(* PLC project Generated.project, CODESYS CODESYS V3.5 SP19 Patch 1 *)
(* stored: creationDateTime 2026-08-18T15:58:33.203512, modificationDateTime 2026-08-18T15:58:33.203512 *)

(* ======================================================================= 🔄 ST_ChainCycleSemiAuto — Diagnostic chronologique Séquenceur Semi-Auto ─────────────────────────────────────────────────────────────── 🎯 Rôle : Vue dépannage / Watch CODESYS pour le cycle semi-automatique 📄 Doc métier : DOC/AF/AF_Partie-14_Fonction_Troubleshooting/FB_TroubleshootingView_v1.2.md 🔒 Sécurité : 100% lecture seule / diagnostic d'observation ======================================================================= *)
TYPE ST_ChainCycleSemiAuto : STRUCT
  Idx101_ModeSemiAutoActive : BOOL;  (* 🚦 1. Conditions d'engagement et autorisations 1 = Mode arbitré SEMI_AUTO actif | 0 = Autre mode *)
  Idx102_PowerAndSafetyOk : BOOL;  (* 1 = Chaîne de sécurité OK (PowerContactorEngaged) *)
  Idx103_HeartbeatIhmOk : BOOL;  (* 1 = Liaison IHM<->PLC valide *)
  Idx104_DeadmanArmed : BOOL;  (* 1 = Bouton homme-mort armé (fenêtre 3s active) *)
  Idx105_MancheDeflechi : BOOL;  (* 1 = Permis mouvement armé (manche hors zone neutre) *)
  Idx106_HomedM1M2 : BOOL;  (* 1 = Codeurs treuils M1 et M2 référencés *)
  Idx107_StartCycleRequest : BOOL;  (* 1 = Demande Start reçue (IHM) *)
  Idx108_AbortCycleRequest : BOOL;  (* 1 = Demande Abort reçue (IHM) *)
  Idx201_Ready : BOOL;  (* 🔄 2. État du Séquenceur 1 = Séquenceur prêt à démarrer *)
  Idx202_Busy : BOOL;  (* 1 = Cycle en cours d'exécution *)
  Idx203_Done : BOOL;  (* 1 = Cycle terminé avec succès *)
  Idx204_Error : BOOL;  (* 1 = Défaut ou anomalie bloquante sur le cycle *)
  Idx205_ErrorId : WORD;  (* Code d'erreur interne FB_Cycle *)
  Idx206_Step : E_CycleStep;  (* Étape courante (X0 à X13 + STABILIZING) *)
  Idx207_StepStr : STRING(40);  (* Libellé explicite de l'étape *)
  Idx208_StepAtError : E_CycleStep;  (* Étape mémorisée lors du dernier défaut *)
  Idx301_TargetPosition : INT;  (* 🎯 3. Consignes & Feedbacks Opérationnels Cible translation sélectionnée (1=Trémie, 3=P1) *)
  Idx302_TargetDepth_M : REAL;  (* Profondeur de consigne (m) *)
  Idx303_KoboldBottomTouch : BOOL;  (* 1 = Détection contact fond Kobold *)
  Idx304_SpeedMismatchActive : BOOL;  (* 1 = Alerte écart de vitesse M1/M2 active *)
  Idx305_LimitLegalReached : BOOL;  (* 1 = Limite légale atteinte (descente bloquée) *)
  Idx306_WinchSyncError : BOOL;  (* 1 = Erreur de synchronisme M1/M2 *)
END_STRUCT;
END_TYPE

(* values of E_CycleStep: X0_PREPARATION: Début de graphe : à la TRÉMIE, treuils en position HAUTE; X1_HOMING: Vitesses lentes pour chercher capteur top + référencement; X2_WORK_POS_SELECT: Sélection cible Trémie/P1/Maintenance + translation validée; X3_OPEN_BUCKET: Ouverture benne (si déjà ouverte -> passe vite); X4_DESCEND_OPEN: Plongée benne ouverte, M1+M2 synchro, Kobold mesure ON; X5_BOTTOM_CONFIRMED: Fond validé (FB_DiveSearch) ; arrêt descente; X6_CLOSE_BUCKET: Fermeture benne — tolérance « à peu près fermé »; X7_CTRL_ASCENT: Remontée palier 1 de contrôle; X8_ASCENT_LOADED: Remontée nominale jusqu'à limite haute; X9_DRAIN_PAUSE: Égouttage temporisé — temps affiché IHM; X10_TRANSLATE_DUMP: Translation vers trémie + avertissements IHM; X11_OPEN_DUMP: Ouverture benne = vidage ; montée possible, descente ouvre; X13_DONE_SYNC: Fin de cycle, synchronisation finale (R4) + compteur; STABILIZING: État d'attente/stabilisation — pas une erreur *)

{attribute 'qualified_only'}
{attribute 'strict'}
TYPE E_CycleStep : (X0_PREPARATION := 0, X1_HOMING := 1, X2_WORK_POS_SELECT := 2, X3_OPEN_BUCKET := 3, X4_DESCEND_OPEN := 4, X5_BOTTOM_CONFIRMED := 5, X6_CLOSE_BUCKET := 6, X7_CTRL_ASCENT := 7, X8_ASCENT_LOADED := 8, X9_DRAIN_PAUSE := 9, X10_TRANSLATE_DUMP := 10, X11_OPEN_DUMP := 11, X13_DONE_SYNC := 13, STABILIZING := 14);
END_TYPE
